(* Logix 5000 project; controller Timers Emulate 5570 rev 33.11; software revision 33.00 *)

TASK T00_MainTask (continuous, watchdog 500 ms) : P00_MainProgram

MODULES
   Local : Emulate 5570 (ICP 2, rev 33.11)
END_MODULES

PROGRAM P00_MainProgram   (* main routine R00_MainRoutine *)
VAR
   B01_Activacion_Alarma : BOOL[32];   // BOOL
   ES : BOOL[32];   // Boton de Paro de emergencia
   I01_Desactivar_Alarma : BOOL[32];   // Boton para desactivar Alarma
   I02_Arranque_Centrifugado : BOOL[32];   // Boton de Arranque del Calentador
   I03_Arranque_Lavadora : BOOL[32];
   I99 : BOOL[32];
   O01_Lampara : BOOL[32];   // Luz de seguridad
   O02_Alarma : BOOL[32];   // Alarma
   O03_Centrifugadora : BOOL[32];   // Encendido de Centrifugadora
   O04_Frenos : BOOL[32];   // Activacion de Frenos
   O05_SegurosPuerta : BOOL[32];   // Activacion de Seguros Puerta
   O06_Lavador : BOOL[32];   // Activacion de Lavadora
   REST : BOOL[32];
   RTO : BOOL[32];
   S01_Movimiento : BOOL[32];   // Sensor de Movimiento
   T01_DesactivarLuz : TIMER[32] := ([0].PRE := 10000, [1].PRE := 10000, [2].PRE := 10000);   // Timer para desactivar luz en 10s
   T02_Alarma : TIMER[32] := ([0].PRE := 5000, [1].PRE := 5000, [2].PRE := 5000);   // Activacion de Alarma
   T03_Centrifugado : TIMER[32] := ([0].PRE := 10000, [2].PRE := 10000);   // Tiempo de centrifugado
   T04_Tiempo_de_Frenado : TIMER[32] := ([0].PRE := 5000, [2].PRE := 5000);   // Tiempo de frenado
   T05_Tiempo_Lavado : TIMER[32] := ([0].PRE := 15000, [1].PRE := 15000);   // Tiempo de Lavado
   T06_Tiempo_Uso : TIMER[32] := ([0].PRE := 60000, [2].PRE := 60000);
   T99_T : TIMER[32] := ([0].PRE := 6000, [0].ACC := 30035);
END_VAR

ROUTINE R00_MainRoutine   (* ladder *)
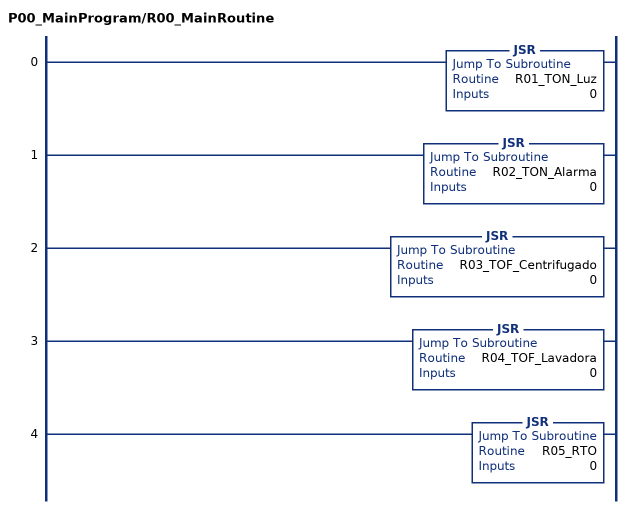
   0: JSR(R01_TON_Luz,0);
   1: JSR(R02_TON_Alarma,0);
   2: JSR(R03_TOF_Centrifugado,0);
   3: JSR(R04_TOF_Lavadora,0);
   4: JSR(R05_RTO,0);
END_ROUTINE

ROUTINE R01_TON_Luz   (* ladder *)
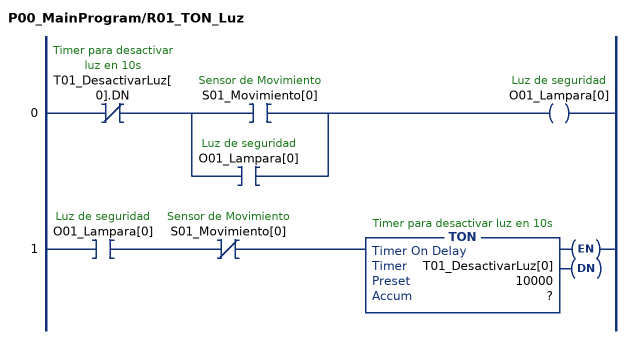
   0: XIO(T01_DesactivarLuz[0].DN)[XIC(S01_Movimiento[0]) ,XIC(O01_Lampara[0]) ]OTE(O01_Lampara[0]);
   1: XIC(O01_Lampara[0])XIO(S01_Movimiento[0])TON(T01_DesactivarLuz[0],?,?);
END_ROUTINE

ROUTINE R02_TON_Alarma   (* ladder *)
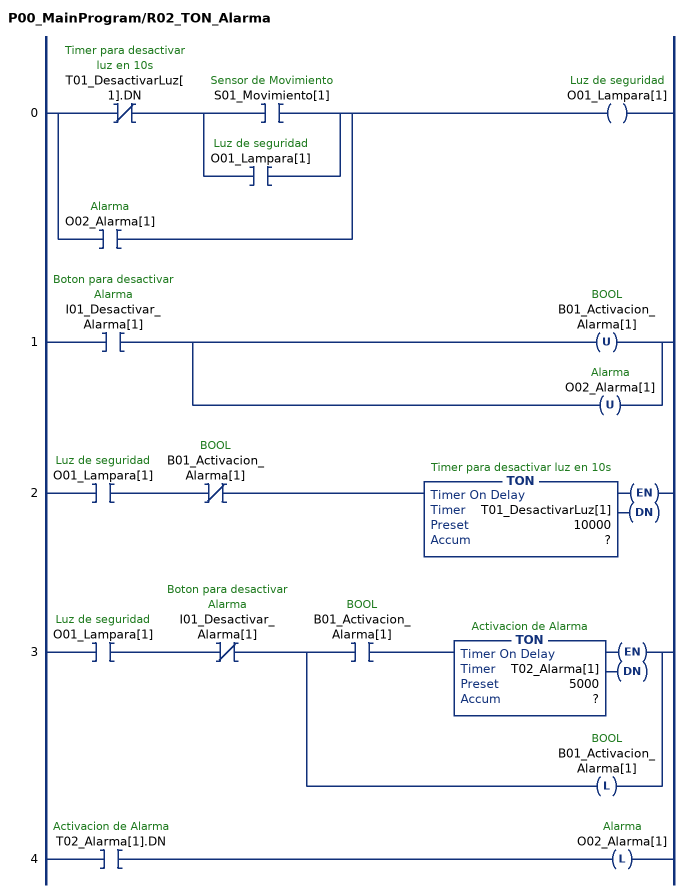
   0: [XIO(T01_DesactivarLuz[1].DN) [XIC(S01_Movimiento[1]) ,XIC(O01_Lampara[1]) ] ,XIC(O02_Alarma[1]) ]OTE(O01_Lampara[1]);
   1: XIC(I01_Desactivar_Alarma[1])[OTU(B01_Activacion_Alarma[1]) ,OTU(O02_Alarma[1]) ];
   2: XIC(O01_Lampara[1])XIO(B01_Activacion_Alarma[1])TON(T01_DesactivarLuz[1],?,?);
   3: XIC(O01_Lampara[1])XIO(I01_Desactivar_Alarma[1])[XIC(B01_Activacion_Alarma[1]) TON(T02_Alarma[1],?,?) ,OTL(B01_Activacion_Alarma[1]) ];
   4: XIC(T02_Alarma[1].DN)OTL(O02_Alarma[1]);
END_ROUTINE

ROUTINE R03_TOF_Centrifugado   (* ladder *)
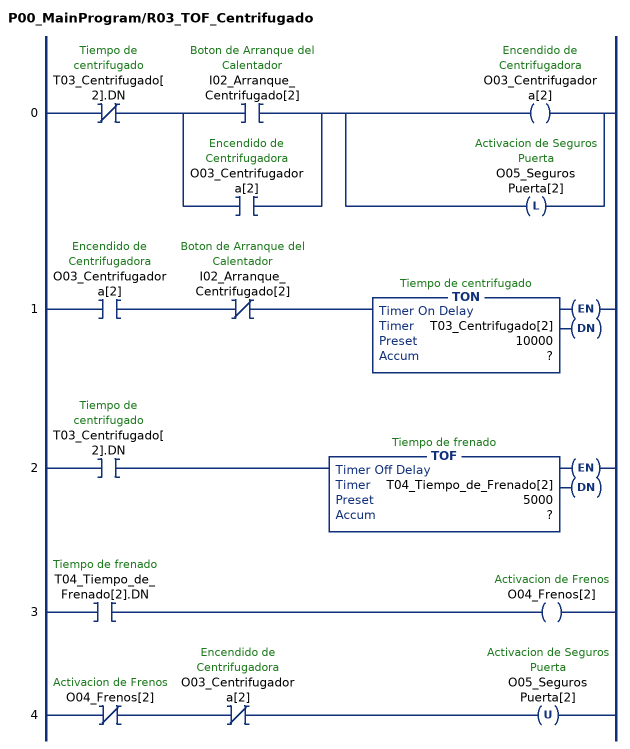
   0: XIO(T03_Centrifugado[2].DN)[XIC(I02_Arranque_Centrifugado[2]) ,XIC(O03_Centrifugadora[2]) ][OTE(O03_Centrifugadora[2]) ,OTL(O05_SegurosPuerta[2]) ];
   1: XIC(O03_Centrifugadora[2])XIO(I02_Arranque_Centrifugado[2])TON(T03_Centrifugado[2],?,?);
   2: XIC(T03_Centrifugado[2].DN)TOF(T04_Tiempo_de_Frenado[2],?,?);
   3: XIC(T04_Tiempo_de_Frenado[2].DN)OTE(O04_Frenos[2]);
   4: XIO(O04_Frenos[2])XIO(O03_Centrifugadora[2])OTU(O05_SegurosPuerta[2]);
END_ROUTINE

ROUTINE R04_TOF_Lavadora   (* ladder *)
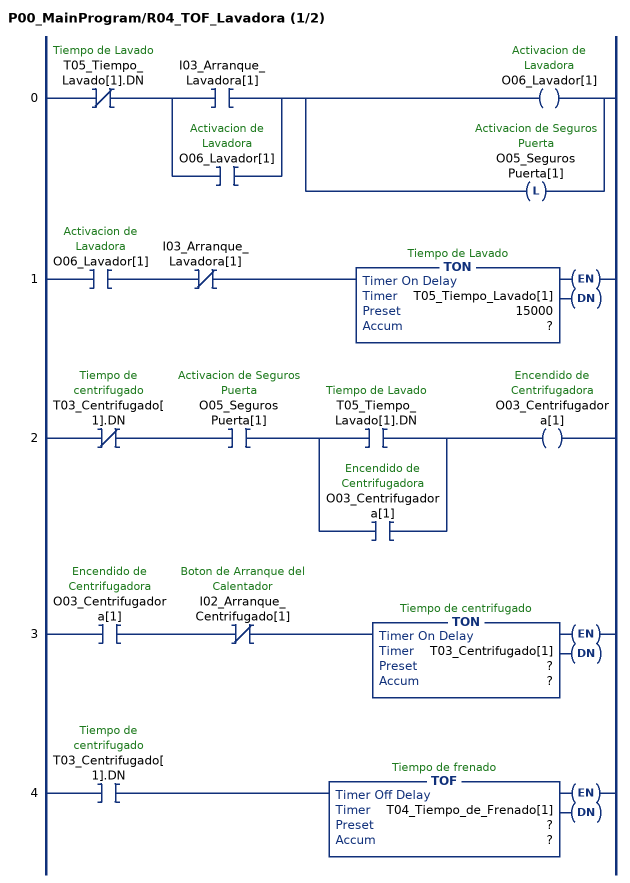
   0: XIO(T05_Tiempo_Lavado[1].DN)[XIC(I03_Arranque_Lavadora[1]) ,XIC(O06_Lavador[1]) ][OTE(O06_Lavador[1]) ,OTL(O05_SegurosPuerta[1]) ];
   1: XIC(O06_Lavador[1])XIO(I03_Arranque_Lavadora[1])TON(T05_Tiempo_Lavado[1],?,?);
   2: XIO(T03_Centrifugado[1].DN)XIC(O05_SegurosPuerta[1])[XIC(T05_Tiempo_Lavado[1].DN) ,XIC(O03_Centrifugadora[1]) ]OTE(O03_Centrifugadora[1]);
   3: XIC(O03_Centrifugadora[1])XIO(I02_Arranque_Centrifugado[1])TON(T03_Centrifugado[1],?,?);
   4: XIC(T03_Centrifugado[1].DN)TOF(T04_Tiempo_de_Frenado[1],?,?);
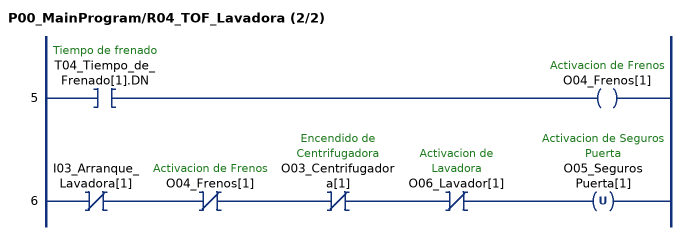
   5: XIC(T04_Tiempo_de_Frenado[1].DN)OTE(O04_Frenos[1]);
   6: XIO(I03_Arranque_Lavadora[1])XIO(O04_Frenos[1])XIO(O03_Centrifugadora[1])XIO(O06_Lavador[1])OTU(O05_SegurosPuerta[1]);
END_ROUTINE

ROUTINE R05_RTO   (* ladder *)
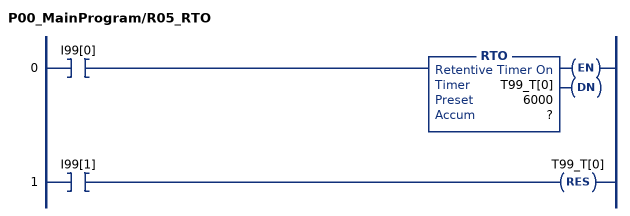
   0: XIC(I99[0])RTO(T99_T[0],?,?);
   1: XIC(I99[1])RES(T99_T[0]);
END_ROUTINE
END_PROGRAM
